// TIA Portal V21 export
DATA_BLOCK "IO BITS"   // DB38
{ S7_Optimized_Access := 'TRUE' }
// stored: MemoryReserve 100
   VAR
      "DOOR1 PRESS BIT" : Bool;   // DOOR1 PRESS BIT
      "DOOR1 VCC BIT" : Bool;   // DOOR1 VCC BIT
      "DOOR2 VCC BIT" : Bool;   // DOOR2 VCC BIT
      "DOOR2 PRESS BIT" : Bool;   // DOOR2 PRESS BIT
      "JACKET SAFETY BIT" : Bool;   // JACKET SAFETY BIT
      "CHAMBER SAFETY BIT" : Bool;   // CHAMBER SAFETY BIT
      PFR : Bool;   // PFR
      "EMG SWITCH" : Bool;   // EMG SWITCH
      "RESET PB" : Bool;   // RESET PB
      "DRUM VFD TRIP" : Bool;   // DRUM VFD TRIP
      "VACCUM PUMP TRIP" : Bool;
      "CRC PUMP TRIP" : Bool;   // CRC PUMP TRIP
      "DOOR1 OPEN LMT" : Bool;   // DOOR1 OPEN LMT
      "DOOR1 CLOSE LMT" : Bool;   // DOOR1 CLOSE LMT
      "DOOR2 OPEN LMT" : Bool;   // DOOR2 OPEN LMT
      "DOOR2 CLOSE LMT" : Bool;   // DOOR2 CLOSE LMT
      "DOOR2 CLOSE PB" : Bool;   // DOOR2 CLOSE PB
      "DOOR2 OPEN PB" : Bool;   // DOOR2 OPEN PB
      "AIR PREESURE SWS" : Bool;   // AIR PREESURE SWS
      "I1.4 SPARE" : Bool;   // I1.4 SPARE
      "I1.5 SPARE" : Bool;   // I1.5 SPARE
      DUMMY : Bool;   // DUMMY
      DUMMY1 : Bool;   // DUMMY1
      "VCC PUMP" : Bool;   // VCC PUMP
      "DOOR1 GASKET" : Bool;   // DOOR1 GASKET
      "CRC MOTOR" : Bool;   // CRC MOTOR
      "JACKET STEAM VAL" : Bool;   // JACKET STEAM VAL
      "CHAMBER STEAM VAL" : Bool;   // CHAMBER STEAM VAL
      "CHAMBER EXHAUST VAL" : Bool;   // CHAMBER EXHAUST VAL
      "CHAMBER VENT VAL" : Bool;   // CHAMBER VENT VAL
      "CHAMBER CONDENSOR VAL" : Bool;   // CHAMBER CONDENSOR VAL
      "WFI VAL" : Bool;   // WFI VAL
      "PWD VAL" : Bool;   // PWD VAL
      "PWD CRC VAL" : Bool;   // PWD CRC VAL
      "DETERGENT DSG VAL" : Bool;   // DETERGENT DSG VAL
      "SILICON DSG VAL" : Bool;   // SILICON DSG VAL
      "DRAIN VAL" : Bool;   // DRAIN VAL
      "DOOR2 INTERLOCK VAL" : Bool;   // DOOR2 INTERLOCK VAL
      "DOOR1 INTERLOCK VAL" : Bool;   // DOOR1 INTERLOCK VAL
      "DOOR1 OPEN VAL" : Bool;   // DOOR1 OPEN VAL
      "DOOR1 CLOSE VAL" : Bool;   // DOOR1 CLOSE VAL
      "DOOR2 OPEN VAL" : Bool;   // DOOR2 OPEN VAL
      "DOOR2 CLOSE VAL" : Bool;   // DOOR2 CLOSE VAL
      "DOOR1 VCC" : Bool;   // DOOR1 VCC
      "DOOR2 GASKET" : Bool;   // DOOR2 GASKET
      "DOOR2 VCC" : Bool;   // DOOR2 VCC
      HOOTER : Bool;   // HOOTER
      "CHAMBER VACCUM VAL" : Bool;
      "CHAMBER STEAM SMALL VAL" : Bool;
      "CHAMBER AIR VENT FAST" : Bool;
      "JACKET STEAM OUT" : Bool;
      "BOW PULSE" : Array[0..100] of Bool;
      "HPHV PULSE" : Array[0..100] of Bool;
      "STANDARD PULSE" : Array[0..100] of Bool;
      "VACUUM PULSE" : Array[0..100] of Bool;
   END_VAR
BEGIN
END_DATA_BLOCK
